// TIA Portal V20 export
FUNCTION "FC_Prueba_1" : Void   // FC1, LAD
{ S7_Optimized_Access := 'TRUE' }
// stored: SetENOAutomatically false
   VAR_INPUT
      ENTRADA_PRUEBA : Bool;
   END_VAR
   VAR_OUTPUT
      SALIDA : Bool;
   END_VAR
BEGIN

REGION Network 1
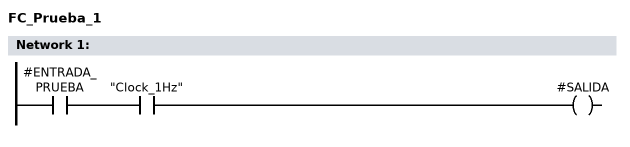
   RUNG wire#powerrail
      Contact( #ENTRADA_PRUEBA )
      Contact( "Clock_1Hz" )
      Coil( #SALIDA )
   END_RUNG
   // the same network as SCL:
   #SALIDA := #ENTRADA_PRUEBA AND "Clock_1Hz";
END_REGION
END_FUNCTION
